PROGRAM MAIN
VAR
	
END_VAR


Encoder.setCounterHorizontal := FALSE;
Encoder.setCounterRotate := FALSE;
Encoder.setCounterVertical := FALSE;

VGR_State();
(*
IF StartStop.IX_START THEN
VGR.QW_VGR_PWM_Vertical_Control := 32;
VGR.QW_VGR_PWM_Vertical_M1 := 3000;
VGR.QX_VGR_M1_VerticalAxisDown_Q2 := TRUE;
ELSIF NOT StartStop.IX_STOP THEN
VGR.QW_VGR_PWM_Vertical_Control := 32;
VGR.QW_VGR_PWM_Vertical_M1 := 3000;
VGR.QX_VGR_M1_VerticalAxisUp_Q1 := TRUE;
ELSE
	VGR.QX_VGR_M1_VerticalAxisUp_Q1 := FALSE;
	VGR.QX_VGR_M1_VerticalAxisDown_Q2 := FALSE;
	VGR.QW_VGR_PWM_Vertical_Control := 0;
VGR.QW_VGR_PWM_Vertical_M1 := 0;
END_IF
*)

END_PROGRAM

(* stored: Version 1.1.0.1, ProductVersion 3.1.4024.12
   POU MAIN: Id {d01eaaea-b107-454d-84d1-9666cf5605a2}, SpecialFunc None *)
